(* PLC project  *)

CONFIGURATION Empty_Module
END_CONFIGURATION
